// Mitsubishi GX Works2 project: PART_REPEAT_SEQUENCE3   PLC: Q03UDV

PROGRAM MAIN
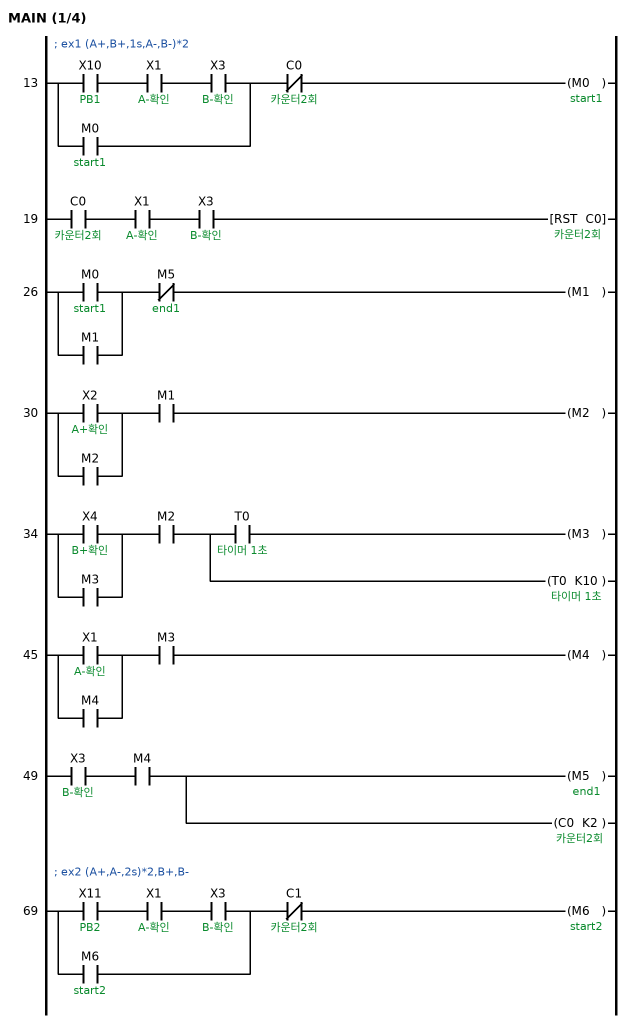
; ex1 (A+,B+,1s,A-,B-)*2
13    LD      X10  ; PB1
      AND     X1  ; A-확인
      AND     X3  ; B-확인
      OR      M0  ; start1
      ANI     C0  ; 카운터2회
      OUT     M0  ; start1
19    LD      C0  ; 카운터2회
      AND     X1  ; A-확인
      AND     X3  ; B-확인
      RST     C0  ; 카운터2회
26    LD      M0  ; start1
      OR      M1
      ANI     M5  ; end1
      OUT     M1
30    LD      X2  ; A+확인
      OR      M2
      AND     M1
      OUT     M2
34    LD      X4  ; B+확인
      OR      M3
      AND     M2
      MPS
      AND     T0  ; 타이머 1초
      OUT     M3
      MPP
      OUT     T0 K10  ; 타이머 1초
45    LD      X1  ; A-확인
      OR      M4
      AND     M3
      OUT     M4
49    LD      X3  ; B-확인
      AND     M4
      OUT     M5  ; end1
      OUT     C0 K2  ; 카운터2회
; ex2 (A+,A-,2s)*2,B+,B-
69    LD      X11  ; PB2
      AND     X1  ; A-확인
      AND     X3  ; B-확인
      OR      M6  ; start2
      ANI     C1  ; 카운터2회
      OUT     M6  ; start2
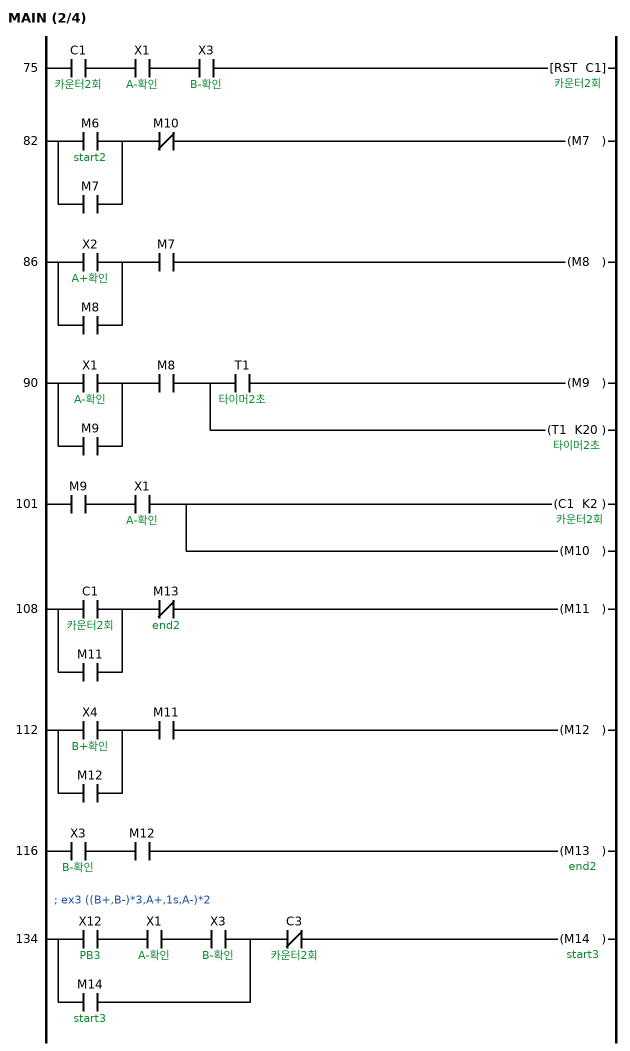
75    LD      C1  ; 카운터2회
      AND     X1  ; A-확인
      AND     X3  ; B-확인
      RST     C1  ; 카운터2회
82    LD      M6  ; start2
      OR      M7
      ANI     M10
      OUT     M7
86    LD      X2  ; A+확인
      OR      M8
      AND     M7
      OUT     M8
90    LD      X1  ; A-확인
      OR      M9
      AND     M8
      MPS
      AND     T1  ; 타이머2초
      OUT     M9
      MPP
      OUT     T1 K20  ; 타이머2초
101   LD      M9
      AND     X1  ; A-확인
      OUT     C1 K2  ; 카운터2회
      OUT     M10
108   LD      C1  ; 카운터2회
      OR      M11
      ANI     M13  ; end2
      OUT     M11
112   LD      X4  ; B+확인
      OR      M12
      AND     M11
      OUT     M12
116   LD      X3  ; B-확인
      AND     M12
      OUT     M13  ; end2
; ex3 ((B+,B-)*3,A+,1s,A-)*2
134   LD      X12  ; PB3
      AND     X1  ; A-확인
      AND     X3  ; B-확인
      OR      M14  ; start3
      ANI     C3  ; 카운터2회
      OUT     M14  ; start3
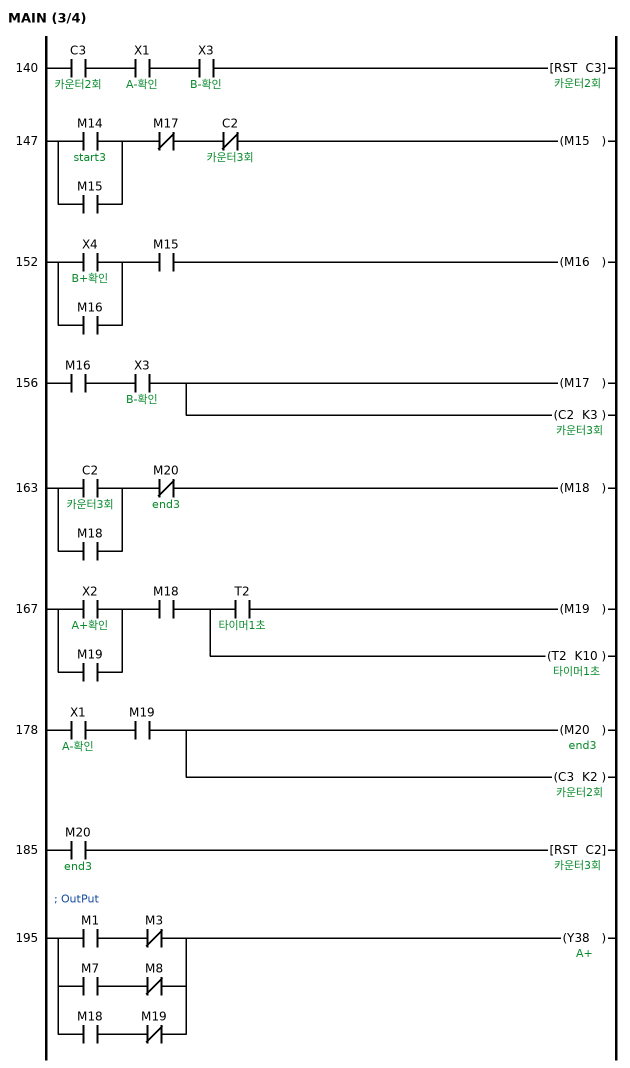
140   LD      C3  ; 카운터2회
      AND     X1  ; A-확인
      AND     X3  ; B-확인
      RST     C3  ; 카운터2회
147   LD      M14  ; start3
      OR      M15
      ANI     M17
      ANI     C2  ; 카운터3회
      OUT     M15
152   LD      X4  ; B+확인
      OR      M16
      AND     M15
      OUT     M16
156   LD      M16
      AND     X3  ; B-확인
      OUT     M17
      OUT     C2 K3  ; 카운터3회
163   LD      C2  ; 카운터3회
      OR      M18
      ANI     M20  ; end3
      OUT     M18
167   LD      X2  ; A+확인
      OR      M19
      AND     M18
      MPS
      AND     T2  ; 타이머1초
      OUT     M19
      MPP
      OUT     T2 K10  ; 타이머1초
178   LD      X1  ; A-확인
      AND     M19
      OUT     M20  ; end3
      OUT     C3 K2  ; 카운터2회
185   LD      M20  ; end3
      RST     C2  ; 카운터3회
; OutPut
195   LD      M1
      ANI     M3
      LD      M7
      ANI     M8
      ORB
      LD      M18
      ANI     M19
      ORB
      OUT     Y38  ; A+
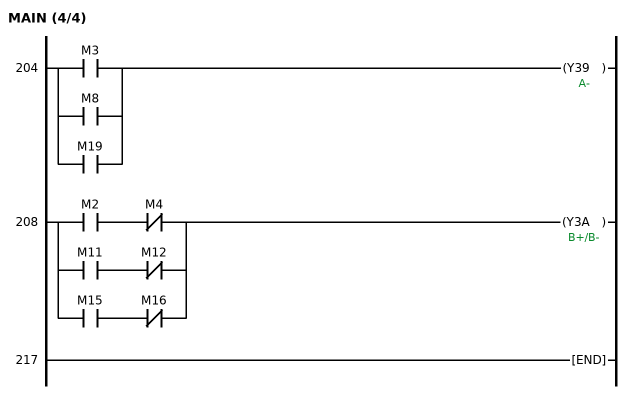
204   LD      M3
      OR      M8
      OR      M19
      OUT     Y39  ; A-
208   LD      M2
      ANI     M4
      LD      M11
      ANI     M12
      ORB
      LD      M15
      ANI     M16
      ORB
      OUT     Y3A  ; B+/B-
217   END
END_PROGRAM
